PROGRAM JIG004_BMW_RAM
VAR
END_VAR

END_PROGRAM

(* stored: Version 1.1.0.1, ProductVersion 3.1.4022.18
   POU JIG004_BMW_RAM: Id {7bf8e275-8f9c-4656-86f8-a1712469daa6}, SpecialFunc None *)
